// TIA Portal V19 export
VAR_GLOBAL   // PLC tag table "Snubber_IO"
   Decoiler1_Snubber_Lift_Ls_UP AT %I125.7 : Bool;   // 712SQ1
   Decoiler1_Snubber_Lift_V_DOWN AT %Q101.4 : Bool;   // 712YV2
   Decoiler1_Snubber_Lift_V_UP AT %Q101.3 : Bool;   // 712YV1
   Decoiler1_Snubber_Roll_V_BWD AT %Q101.5 : Bool;   // 712YV3
   Decoiler1_Snubber_Roll_V_FWD AT %Q101.6 : Bool;   // 712YV4
   Decoiler2_Snubber_Lift_Ls_UP AT %I126.2 : Bool;   // 717SQ1
   Decoiler2_Snubber_Lift_V_DOWN AT %Q102.4 : Bool;   // 717YV2
   Decoiler2_Snubber_Lift_V_UP AT %Q102.3 : Bool;   // 717YV1
   Decoiler2_Snubber_Roll_V_BWD AT %Q102.5 : Bool;   // 717YV3
   Decoiler2_Snubber_Roll_V_FWD AT %Q102.6 : Bool;   // 717YV4
END_VAR
